PROGRAM MAIN
VAR
END_VAR

mictestonetwo();

END_PROGRAM

(* stored: Version 1.1.0.1, ProductVersion 3.1.4024.12
   POU MAIN: Id {73494d6d-a9c9-4353-aeaf-36b72084351a}, SpecialFunc None *)
